// TIA Portal V21 export
// export: Created 2026-09-06T18:39:46.6337555Z, ExportSetting WithDefaults, DisplayName Totally Integrated Automation Portal, DisplayVersion V21 Hotfix 1, DisplayName STEP 7 Professional, DisplayVersion V21, DisplayName STEP 7 CFC, DisplayVersion V21, DisplayName STEP 7 Safety, DisplayVersion V21, DisplayName Tech WebApplication, DisplayVersion V21, DisplayName WinCC Basic/Comfort/Advanced, DisplayVersion V21, DisplayName SIMATIC Visualization Architect, DisplayVersion V21, DisplayName WinCC Unified, DisplayVersion V21, DisplayName SIMATIC Visualization Architect, DisplayVersion V21
VAR_GLOBAL   // PLC tag table "Entradas_Expansao1_SM1221"
   SIN_Y7_COMP AT %I2.0 : Bool;   // Diagnostico de Seguranca do Compactador (Rele IFM Y7)
   NA_S1_COMP AT %I2.1 : Bool;   // Interlock / Fim de Curso de Seguranca 1 do Compactador
   NA_S2_COMP AT %I2.2 : Bool;   // Interlock / Fim de Curso de Seguranca 2 do Compactador
   NA_S3_COMP AT %I2.3 : Bool;   // Interlock / Fim de Curso de Seguranca 3 do Compactador
   SIN_Y7_M1 AT %I2.4 : Bool;   // Diagnostico de Seguranca do Motor M1 (Rele IFM Y7)
   NA_STOP_M1 AT %I2.5 : Bool;   // Botao / Paragem Local de Seguranca do Tapete M1
   SIN_Y7_M2 AT %I2.6 : Bool;   // Diagnostico de Seguranca do Motor M2 (Rele IFM Y7)
   SIN_Y7_M3 AT %I2.7 : Bool;   // Diagnostico de Seguranca do Motor M3 (Rele IFM Y7)
   NA_STOP_M2 AT %I3.0 : Bool;   // Botao / Paragem Local de Seguranca do Tapete M2
   NA_STOP_M3 AT %I3.1 : Bool;   // Botao / Paragem Local de Seguranca do Tapete M3
   SIN_Y7_M4 AT %I3.2 : Bool;   // Diagnostico de Seguranca do Motor M4 (Rele IFM Y7)
   NA_STOP_M4 AT %I3.3 : Bool;   // Botao / Paragem Local de Seguranca do Tapete M4
   SIN_Y7_M5 AT %I3.4 : Bool;   // Diagnostico de Seguranca do Motor M5 (Rele IFM Y7)
   NA_STOP_M5 AT %I3.5 : Bool;   // Botao / Paragem Local de Seguranca do Tapete M5
   SENSOR_75_PERCENT AT %I3.6 : Bool;   // Sensor Optoeletronico de Nivel da Moega a 75%
   SENSOR_100_PERCENT AT %I3.7 : Bool;   // Sensor Optoeletronico de Nivel da Moega a 100%
END_VAR
